TYPE CuBaseRecurringFailures EXTENDS TcoCore.TcoStruct : 
	STRUCT
   		ArbitrarilyRecurringFails : CuBaseRecurringFail;
    	SameRecurringFails : CuBaseRecurringFail;
	END_STRUCT
END_TYPE

(* stored: Version 1.1.0.1
   DUT CuBaseRecurringFailures: Id {9c9d3c5b-f8e2-04ee-0d59-7c39ee743c2d} *)
